Staubli VAL3: moveRobot.pgx

program moveRobot(point x_pMoveTo (dimensions=1))
  local bool l_bResult
  local joint l_jMoveTo
  local num l_nValue[3]
  local point l_pMoveTo
begin
  nMotionError=0
  // Check if destination is reachabled
  l_pMoveTo=appro(here(tPointer,world),cfg:trApproach)
  l_bResult=pointToJoint(tPointer,herej(),l_pMoveTo,l_jMoveTo)
  if l_bResult==true
    movel(l_pMoveTo,tPointer,mSlow)
    l_pMoveTo=appro(x_pMoveTo,cfg:trApproach)
    l_bResult=pointToJoint(tPointer,herej(),l_pMoveTo,l_jMoveTo)
    if l_bResult==true
      movej(l_pMoveTo,tPointer,mSlow)
      l_pMoveTo=x_pMoveTo
      l_bResult=pointToJoint(tPointer,herej(),l_pMoveTo,l_jMoveTo)
      if l_bResult==true
        movel(x_pMoveTo,tPointer,mSlow)
      else
        nMotionError=55
      endIf
    else
      nMotionError=54
    endIf
  else
    nMotionError=53
  endIf
  // Prepare clear text error message
  if nMotionError!=0
    l_nValue[0]=cfg:trApproach.x
    l_nValue[1]=cfg:trApproach.y
    l_nValue[2]=cfg:trApproach.z
    call ut:addNumToString(lang:sListOfMessage[nMotionError],sErrorMessage,"*",l_nValue)
  endIf
end
